// Mitsubishi GX Works2 project: PLC 카운터   PLC: Q03UDV

PROGRAM MAIN
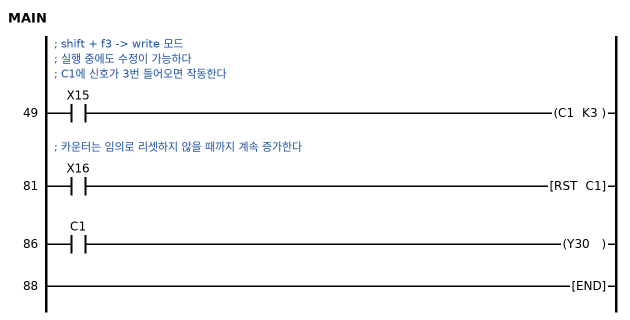
; shift + f3 -> write 모드
; 실행 중에도 수정이 가능하다
; C1에 신호가 3번 들어오면 작동한다
49    LD      X15
      OUT     C1 K3
; 카운터는 임의로 리셋하지 않을 때까지 계속 증가한다
81    LD      X16
      RST     C1
86    LD      C1
      OUT     Y30
88    END
END_PROGRAM
